(* Logix 5000 project; controller cal1615 1756-L62 rev 20.19; software revision 20.05; part 33 of 81 *)
(* tags used below, declared in another part *)
   FAULT : BOOL;   // Fault AFI
   p01_param_fan_zero_speed : REAL;
   p01_param_open_oven_recirc_sp : REAL;
   p01_recipe_active : recipe;   // Active Recipe
   p01_sys_scp : SYS_SCP;   // System Scaling
   p01r09_open_oven : BOOL;
   p01r09_pb_global_reset : BOOL;   // System Modes PB: Global Fault Reset
   p02_dint_from_hmi : hmi_dint;
   p11r02_shutdown_temp : BOOL;   // Zone 1 Misc Control Safe Shutdown Temperature
   p11r30 : routine;   // Zone 1 Temperature Control
   p12r02_shutdown_temp : BOOL;   // Zone 2 Misc Control Safe Shutdown Temperature
   p12r30 : routine;   // Zone 2 Temperature Control
   p13_ai_recirc_rpm : REAL;   // Zone 3 Analog Input Recirc Fan RPM
   p13_ao_recirc_selected_speed : REAL;   // Zone 3 Analog Output Recirc Fan VFD Selected Speed
   p13_di_recirc : acs800_di_normal;   // Zone 3 Digital Inputs Recirc Fan
   p13_di_recirc_fan_mtr_ts : BOOL;   // Zone 3 Digital Input Recirc Fan Motor Thermostat OK
   p13_di_recirc_flow_ok : BOOL;   // Zone 3 Digital Input Recirc Flow OK
   p13_dint_to_hmi : DINT[16];   // Zone 3 Temperature Control VFDs On
   p13_do_recirc : acs800_do_normal;   // Zone 3 Digital Outputs Supply Fan
   p13r01 : routine;   // Zone 3 Main
   p13r02_shutdown_temp : BOOL;   // Zone 3 Misc Control Safe Shutdown Temperature
   p13r20_state : DINT;   // Zone 3 Temperature Control State
   p13r32 : routine;   // Zone 3 Recirc VFD
   p13r32_pb_start : BOOL;   // Zone 3 Recirc VFD PB: Start
   p13r32_pb_stop : BOOL;   // Zone 3 Recirc VFD PB: Stop
   p13r32_request_auto_run : BOOL;   // Zone 3 Recirc Fan Run Request
   p13r32_run_permissive : BOOL;   // Zone 3 Recirc VFD Run Permissive
   p13r32_timer_fault : TIMER[5];   // Zone 3 Recirc VFD Fault Timer
   p13r32_timer_warning : TIMER[5];   // Zone 3 Supply VFD Warning Timer
   p13r32_vfd_stopped : BOOL;   // Zone 3 Recirc VFD VFD Stopped
   p19_ai_prs : REAL;   // Advanced Cooling Analog Input Pressure [PSI]
   p19_ai_tc01 : REAL;   // Advanced Cooling Analog Input Control Temperature 1
   p19_di_pump : BOOL;
   p19_di_tc01_bo : BOOL;   // Advanced Cooling Digital Input Control Thermocouple 1 Failure
   p19_di_tc02_bo : BOOL;   // Advanced Cooling Digital Input Control Thermocouple 2 Failure
   p19_dint_to_hmi : DINT[16];
   p19_param_tc01z : REAL;   // Advanced Cooling Parameter Control Temperature 1 Zero Offset
   p19r01 : routine;   // Advanced Cooling Main
   p19r02 : routine;   // Advanced Cooling Misc Control
   p19r02_fault_exists : BOOL;
   p19r02_timer_fault : TIMER[4];   // Advanced Cooling Misc Control Fault Delay
   p19r02_timer_warning : TIMER[4];   // Advanced Cooling Warning Delay
   p19r02_unack_fault : BOOL;   // Advanced Cooling Misc Control Unacknowledged Fault
   p19r02_unack_warning : BOOL;   // Advanced Cooling Misc Control Unacknowledged Warning
   p19r02_warning_exists : BOOL;
   p19r03 : routine;   // Advanced Cooling Input
   p19r03_prs_input_max : REAL;
   p19r03_prs_input_min : REAL;
   p19r03_prs_output_max : REAL;
   p19r03_prs_output_min : REAL;
   p19r03_timer_fault : TIMER[4];   // Advanced Cooling Input
   p19r03_timer_warning : TIMER[4];   // Advanced Cooling Input
   p19r04 : routine;   // Advanced Cooling Output
   p19r05 : routine;   // Advanced Cooling Dint to HMI
   p19r06 : routine;   // Advanced Cooling Real to HMI
   p19r07 : routine;   // Advanced Cooling Alarms
   p19r08 : routine;   // Advanced Cooling Warnings
   p19r09 : routine;   // Advanced Cooling Modes
   p19r10 : routine;   // Advanced Cooling Parameters
   p19r30 : routine;   // Advanced Cooling Temperature Control
   p19r31 : routine;   // Advanced Cooling Pump
   p23r02 : routine;   // Impreg Misc Control
(* P13_Zone_3, continued *)

ROUTINE R32_Recirc_VFD   (* ladder *)
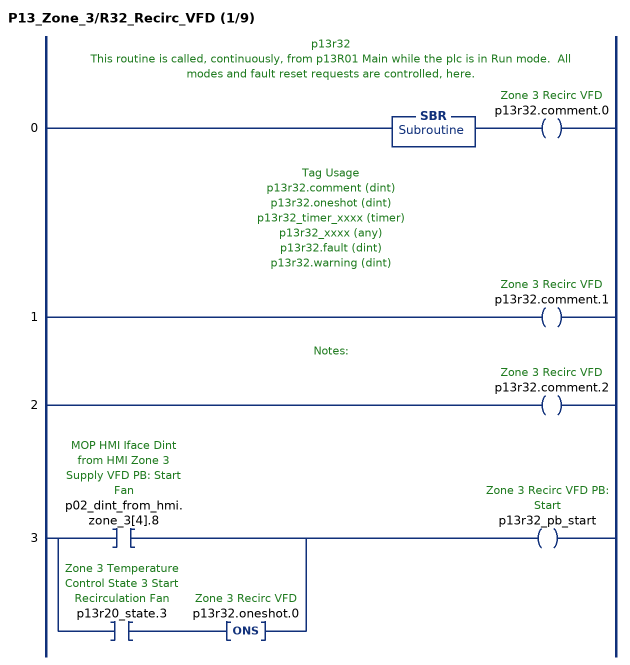
   // p13r32
   // This routine is called, continuously, from p13R01 Main while the plc is in Run mode.  All modes and fault reset requests are controlled, here.
   0: SBR()OTE(p13r32.comment.0);
   // Tag Usage
   // p13r32.comment (dint)
   // p13r32.oneshot (dint)
   // p13r32_timer_xxxx (timer)
   // p13r32_xxxx (any)
   // p13r32.fault (dint)
   // p13r32.warning (dint)
   1: OTE(p13r32.comment.1);
   // Notes:
   2: OTE(p13r32.comment.2);
   3: [XIC(p02_dint_from_hmi.zone_3[4].8) ,XIC(p13r20_state.3) ONS(p13r32.oneshot.0) ]OTE(p13r32_pb_start);
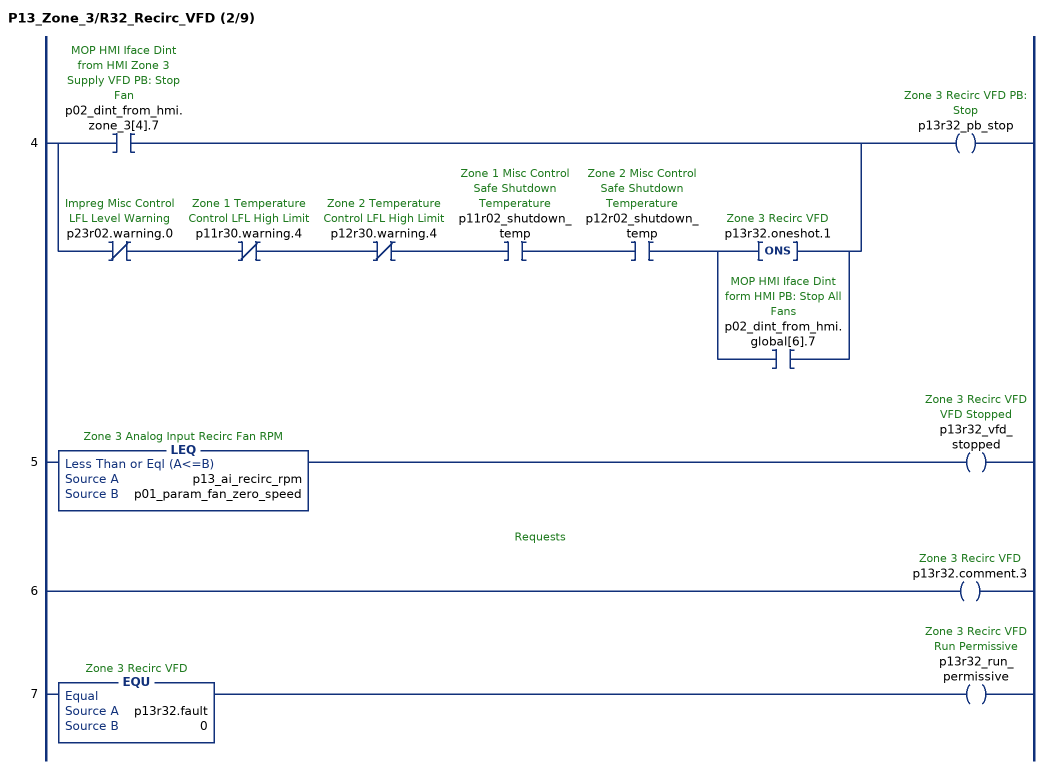
   4: [XIC(p02_dint_from_hmi.zone_3[4].7) ,XIO(p23r02.warning.0) XIO(p11r30.warning.4) XIO(p12r30.warning.4) XIC(p11r02_shutdown_temp) XIC(p12r02_shutdown_temp) [ONS(p13r32.oneshot.1) ,XIC(p02_dint_from_hmi.global[6].7) ] ]OTE(p13r32_pb_stop);
   5: LEQ(p13_ai_recirc_rpm,p01_param_fan_zero_speed)OTE(p13r32_vfd_stopped);
   // Requests
   6: OTE(p13r32.comment.3);
   7: EQU(p13r32.fault,0)OTE(p13r32_run_permissive);
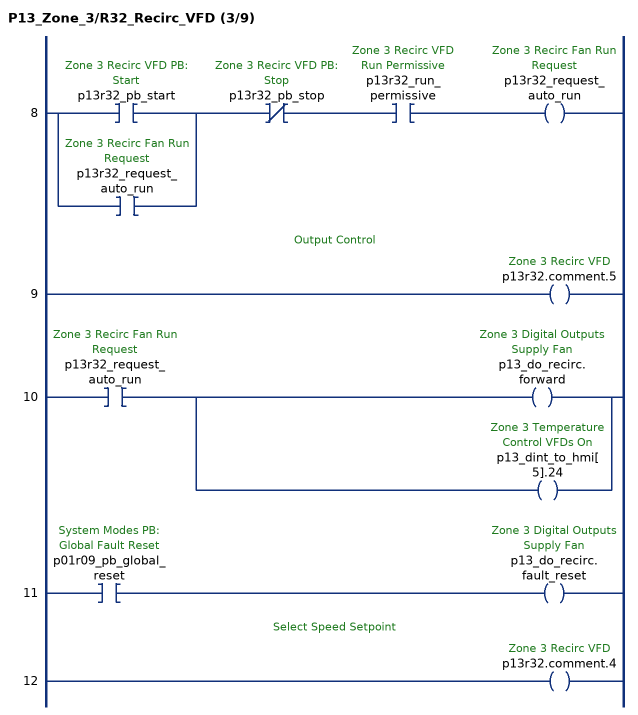
   8: [XIC(p13r32_pb_start) ,XIC(p13r32_request_auto_run) ]XIO(p13r32_pb_stop)XIC(p13r32_run_permissive)OTE(p13r32_request_auto_run);
   // Output Control
   9: OTE(p13r32.comment.5);
   10: XIC(p13r32_request_auto_run)[OTE(p13_do_recirc.forward) ,OTE(p13_dint_to_hmi[5].24) ];
   11: XIC(p01r09_pb_global_reset)OTE(p13_do_recirc.fault_reset);
   // Select Speed Setpoint
   12: OTE(p13r32.comment.4);
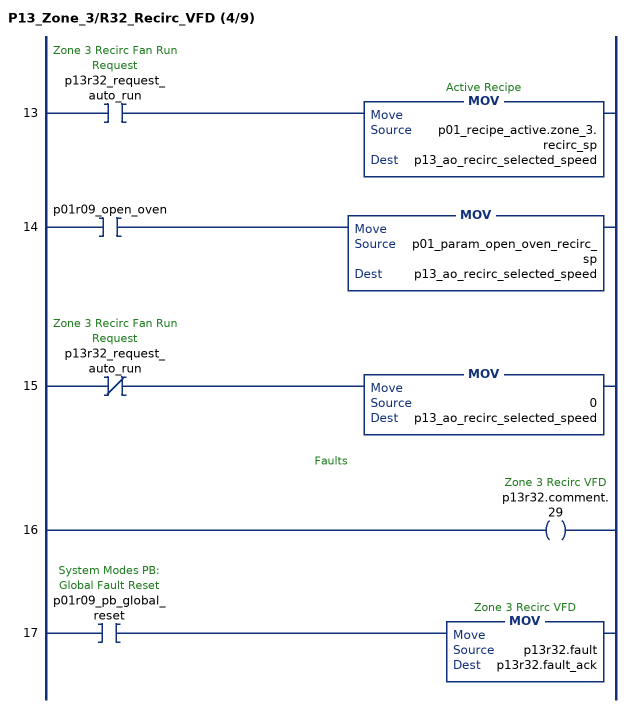
   13: XIC(p13r32_request_auto_run)MOV(p01_recipe_active.zone_3.recirc_sp,p13_ao_recirc_selected_speed);
   14: XIC(p01r09_open_oven)MOV(p01_param_open_oven_recirc_sp,p13_ao_recirc_selected_speed);
   15: XIO(p13r32_request_auto_run)MOV(0,p13_ao_recirc_selected_speed);
   // Faults
   16: OTE(p13r32.comment.29);
   17: XIC(p01r09_pb_global_reset)MOV(p13r32.fault,p13r32.fault_ack);
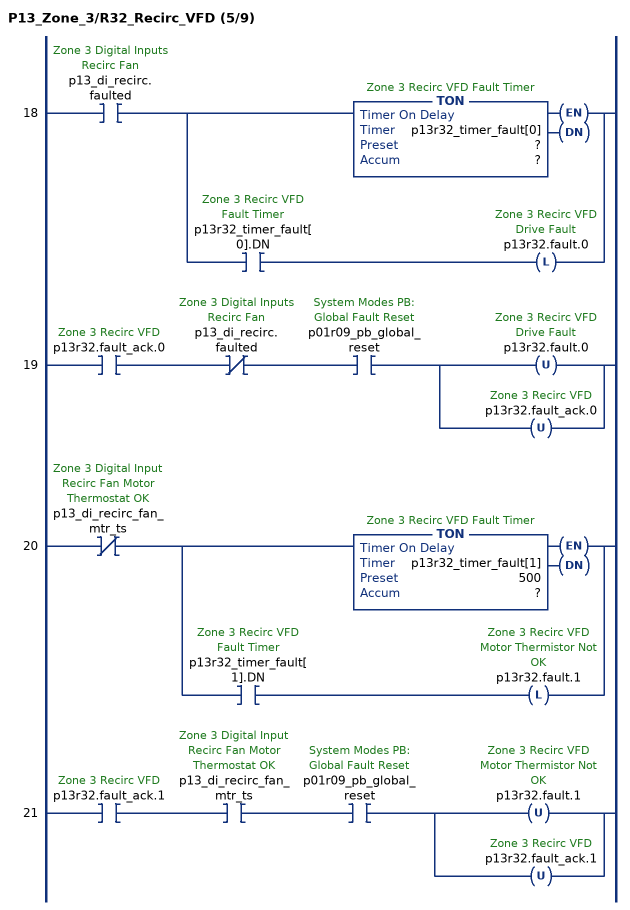
   18: XIC(p13_di_recirc.faulted)[TON(p13r32_timer_fault[0],?,?) ,XIC(p13r32_timer_fault[0].DN) OTL(p13r32.fault.0) ];
   19: XIC(p13r32.fault_ack.0)XIO(p13_di_recirc.faulted)XIC(p01r09_pb_global_reset)[OTU(p13r32.fault.0) ,OTU(p13r32.fault_ack.0) ];
   20: XIO(p13_di_recirc_fan_mtr_ts)[TON(p13r32_timer_fault[1],?,?) ,XIC(p13r32_timer_fault[1].DN) OTL(p13r32.fault.1) ];
   21: XIC(p13r32.fault_ack.1)XIC(p13_di_recirc_fan_mtr_ts)XIC(p01r09_pb_global_reset)[OTU(p13r32.fault.1) ,OTU(p13r32.fault_ack.1) ];
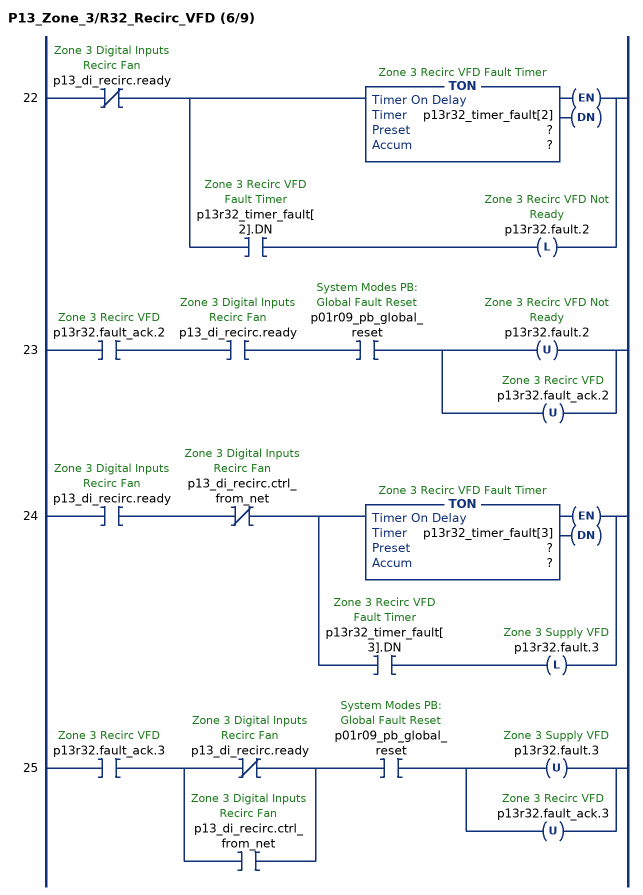
   22: XIO(p13_di_recirc.ready)[TON(p13r32_timer_fault[2],?,?) ,XIC(p13r32_timer_fault[2].DN) OTL(p13r32.fault.2) ];
   23: XIC(p13r32.fault_ack.2)XIC(p13_di_recirc.ready)XIC(p01r09_pb_global_reset)[OTU(p13r32.fault.2) ,OTU(p13r32.fault_ack.2) ];
   24: XIC(p13_di_recirc.ready)XIO(p13_di_recirc.ctrl_from_net)[TON(p13r32_timer_fault[3],?,?) ,XIC(p13r32_timer_fault[3].DN) OTL(p13r32.fault.3) ];
   25: XIC(p13r32.fault_ack.3)[XIO(p13_di_recirc.ready) ,XIC(p13_di_recirc.ctrl_from_net) ]XIC(p01r09_pb_global_reset)[OTU(p13r32.fault.3) ,OTU(p13r32.fault_ack.3) ];
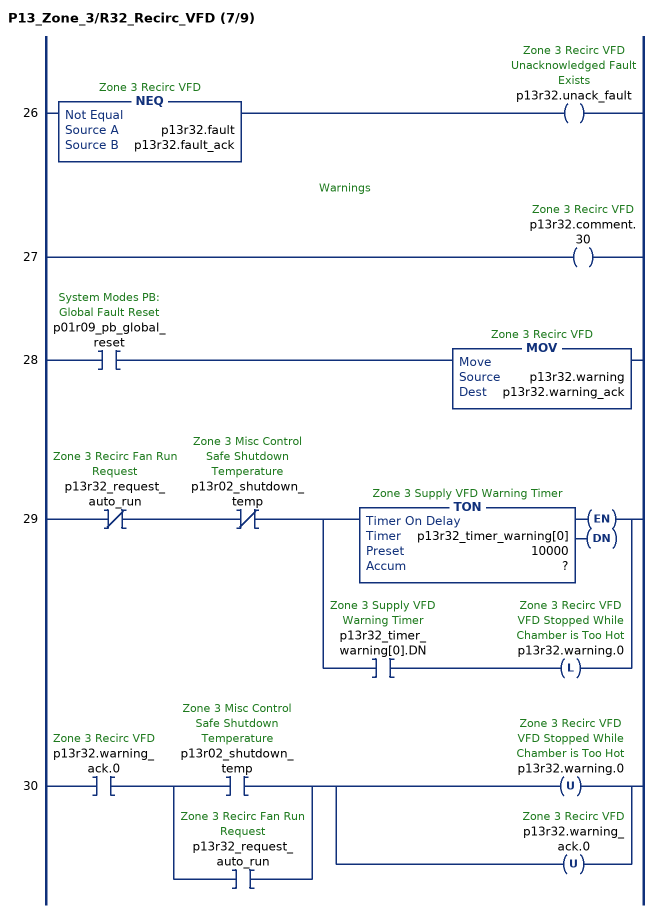
   26: NEQ(p13r32.fault,p13r32.fault_ack)OTE(p13r32.unack_fault);
   // Warnings
   27: OTE(p13r32.comment.30);
   28: XIC(p01r09_pb_global_reset)MOV(p13r32.warning,p13r32.warning_ack);
   29: XIO(p13r32_request_auto_run)XIO(p13r02_shutdown_temp)[TON(p13r32_timer_warning[0],?,?) ,XIC(p13r32_timer_warning[0].DN) OTL(p13r32.warning.0) ];
   30: XIC(p13r32.warning_ack.0)[XIC(p13r02_shutdown_temp) ,XIC(p13r32_request_auto_run) ][OTU(p13r32.warning.0) ,OTU(p13r32.warning_ack.0) ];
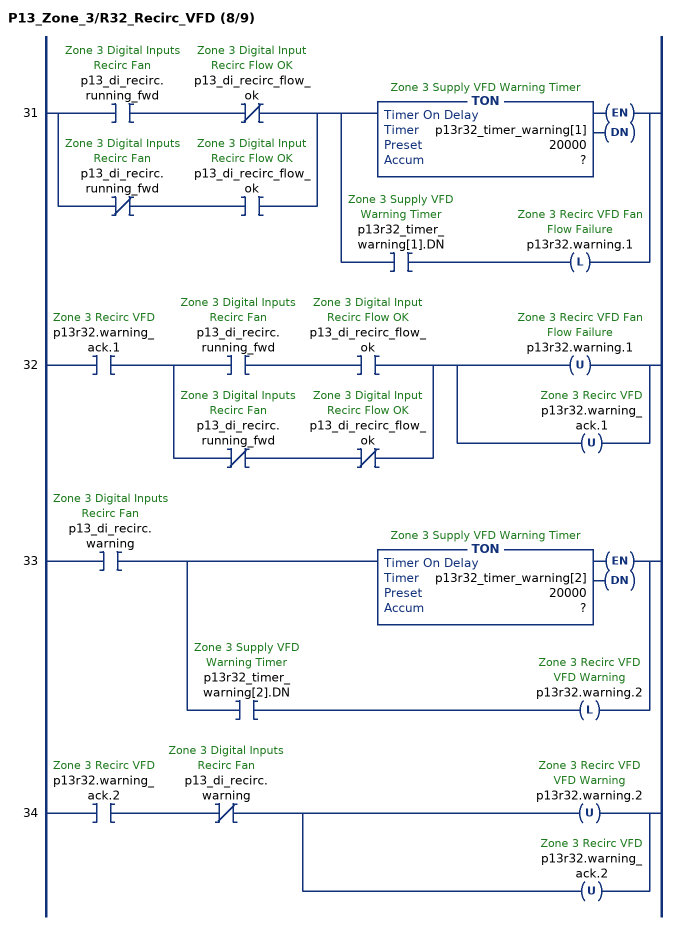
   31: [XIC(p13_di_recirc.running_fwd) XIO(p13_di_recirc_flow_ok) ,XIO(p13_di_recirc.running_fwd) XIC(p13_di_recirc_flow_ok) ][TON(p13r32_timer_warning[1],?,?) ,XIC(p13r32_timer_warning[1].DN) OTL(p13r32.warning.1) ];
   32: XIC(p13r32.warning_ack.1)[XIC(p13_di_recirc.running_fwd) XIC(p13_di_recirc_flow_ok) ,XIO(p13_di_recirc.running_fwd) XIO(p13_di_recirc_flow_ok) ][OTU(p13r32.warning.1) ,OTU(p13r32.warning_ack.1) ];
   33: XIC(p13_di_recirc.warning)[TON(p13r32_timer_warning[2],?,?) ,XIC(p13r32_timer_warning[2].DN) OTL(p13r32.warning.2) ];
   34: XIC(p13r32.warning_ack.2)XIO(p13_di_recirc.warning)[OTU(p13r32.warning.2) ,OTU(p13r32.warning_ack.2) ];
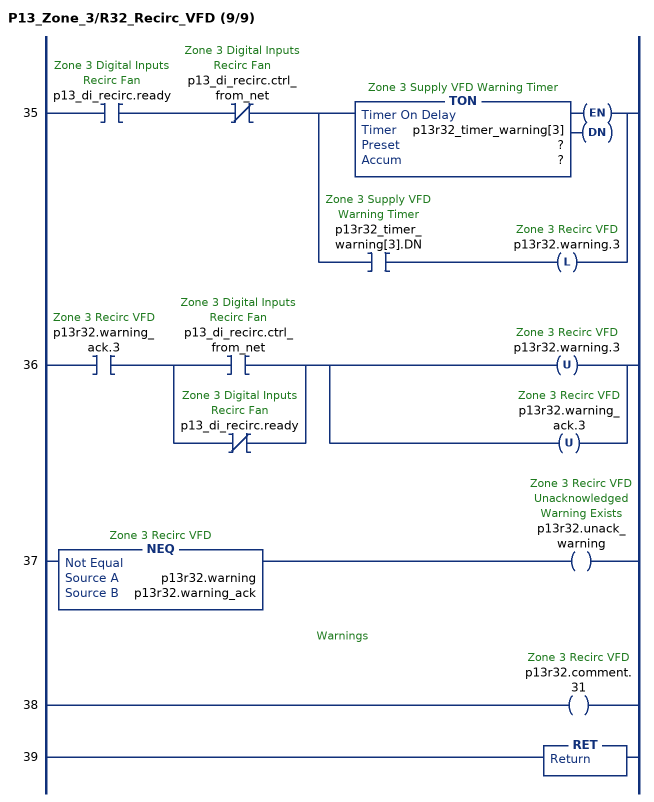
   35: XIC(p13_di_recirc.ready)XIO(p13_di_recirc.ctrl_from_net)[TON(p13r32_timer_warning[3],?,?) ,XIC(p13r32_timer_warning[3].DN) OTL(p13r32.warning.3) ];
   36: XIC(p13r32.warning_ack.3)[XIC(p13_di_recirc.ctrl_from_net) ,XIO(p13_di_recirc.ready) ][OTU(p13r32.warning.3) ,OTU(p13r32.warning_ack.3) ];
   37: NEQ(p13r32.warning,p13r32.warning_ack)OTE(p13r32.unack_warning);
   // Warnings
   38: OTE(p13r32.comment.31);
   39: RET();
END_ROUTINE
END_PROGRAM

PROGRAM P19_Advanced_Cooling   (* main routine R01_Main *)

ROUTINE R01_Main   (* ladder *)
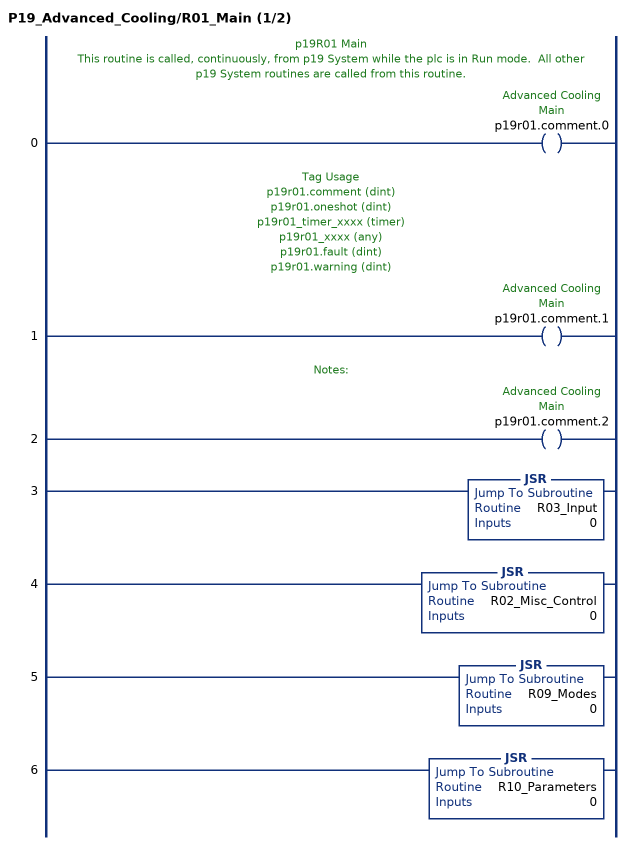
   // p19R01 Main
   // This routine is called, continuously, from p19 System while the plc is in Run mode.  All other p19 System routines are called from this routine.
   0: OTE(p19r01.comment.0);
   // Tag Usage
   // p19r01.comment (dint)
   // p19r01.oneshot (dint)
   // p19r01_timer_xxxx (timer)
   // p19r01_xxxx (any)
   // p19r01.fault (dint)
   // p19r01.warning (dint)
   1: OTE(p19r01.comment.1);
   // Notes:
   2: OTE(p19r01.comment.2);
   3: JSR(R03_Input,0);
   4: JSR(R02_Misc_Control,0);
   5: JSR(R09_Modes,0);
   6: JSR(R10_Parameters,0);
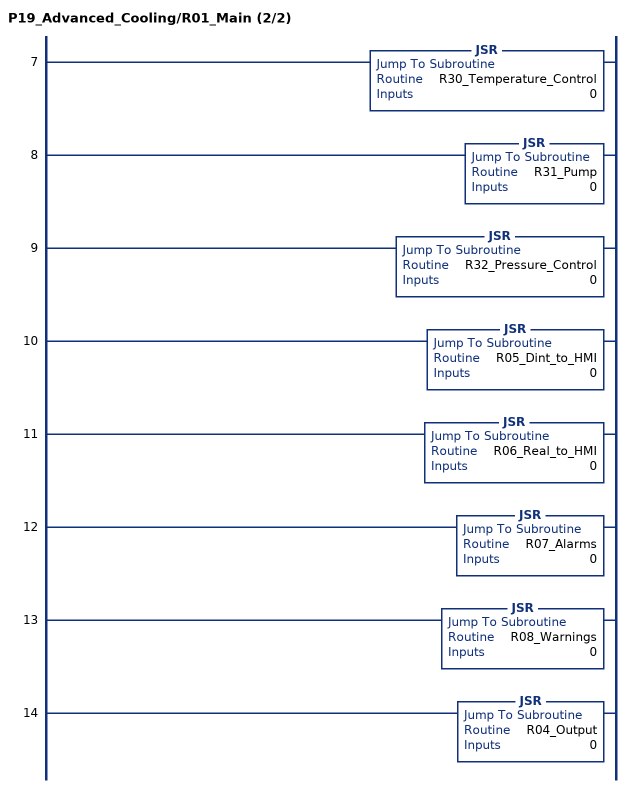
   7: JSR(R30_Temperature_Control,0);
   8: JSR(R31_Pump,0);
   9: JSR(R32_Pressure_Control,0);
   10: JSR(R05_Dint_to_HMI,0);
   11: JSR(R06_Real_to_HMI,0);
   12: JSR(R07_Alarms,0);
   13: JSR(R08_Warnings,0);
   14: JSR(R04_Output,0);
END_ROUTINE

ROUTINE R02_Misc_Control   (* ladder *)
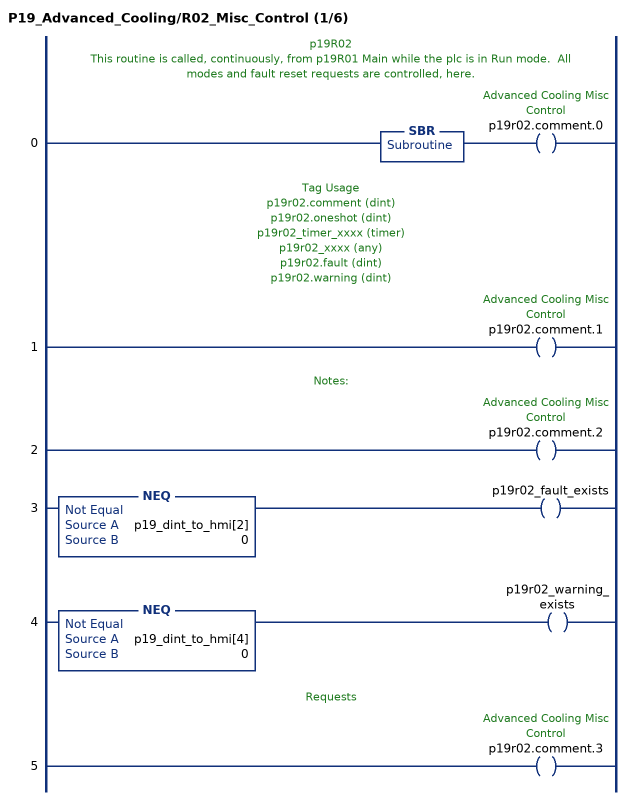
   // p19R02
   // This routine is called, continuously, from p19R01 Main while the plc is in Run mode.  All modes and fault reset requests are controlled, here.
   0: SBR()OTE(p19r02.comment.0);
   // Tag Usage
   // p19r02.comment (dint)
   // p19r02.oneshot (dint)
   // p19r02_timer_xxxx (timer)
   // p19r02_xxxx (any)
   // p19r02.fault (dint)
   // p19r02.warning (dint)
   1: OTE(p19r02.comment.1);
   // Notes:
   2: OTE(p19r02.comment.2);
   3: NEQ(p19_dint_to_hmi[2],0)OTE(p19r02_fault_exists);
   4: NEQ(p19_dint_to_hmi[4],0)OTE(p19r02_warning_exists);
   // Requests
   5: OTE(p19r02.comment.3);
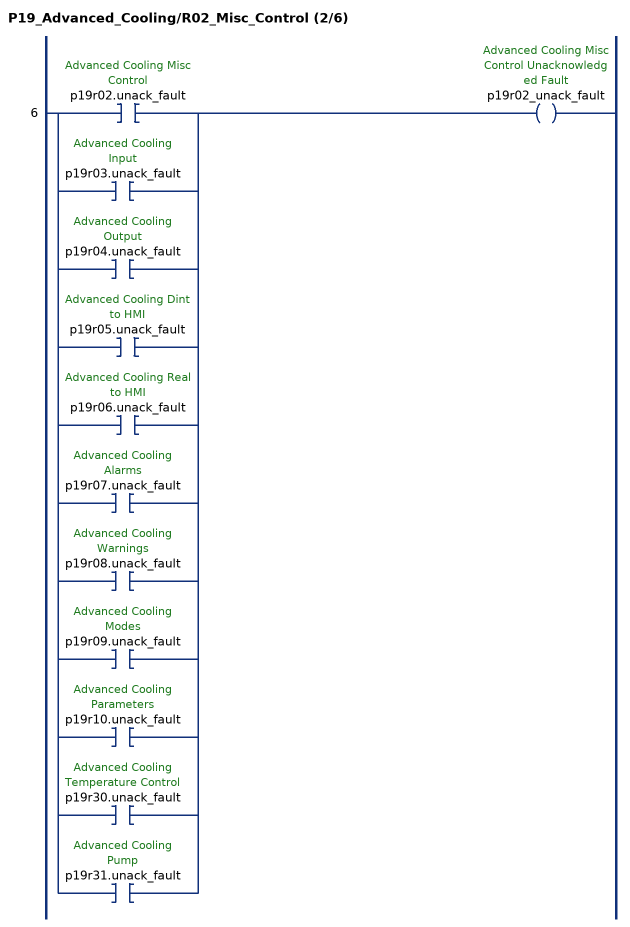
   6: [XIC(p19r02.unack_fault) ,XIC(p19r03.unack_fault) ,XIC(p19r04.unack_fault) ,XIC(p19r05.unack_fault) ,XIC(p19r06.unack_fault) ,XIC(p19r07.unack_fault) ,XIC(p19r08.unack_fault) ,XIC(p19r09.unack_fault) ,XIC(p19r10.unack_fault) ,XIC(p19r30.unack_fault) ,XIC(p19r31.unack_fault) ]OTE(p19r02_unack_fault);
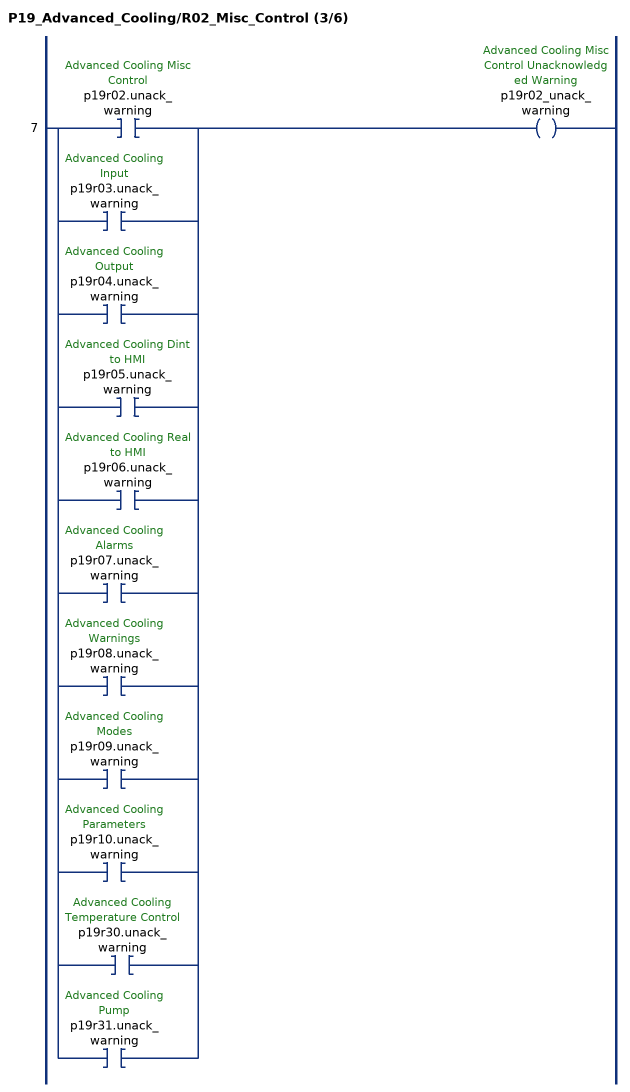
   7: [XIC(p19r02.unack_warning) ,XIC(p19r03.unack_warning) ,XIC(p19r04.unack_warning) ,XIC(p19r05.unack_warning) ,XIC(p19r06.unack_warning) ,XIC(p19r07.unack_warning) ,XIC(p19r08.unack_warning) ,XIC(p19r09.unack_warning) ,XIC(p19r10.unack_warning) ,XIC(p19r30.unack_warning) ,XIC(p19r31.unack_warning) ]OTE(p19r02_unack_warning);
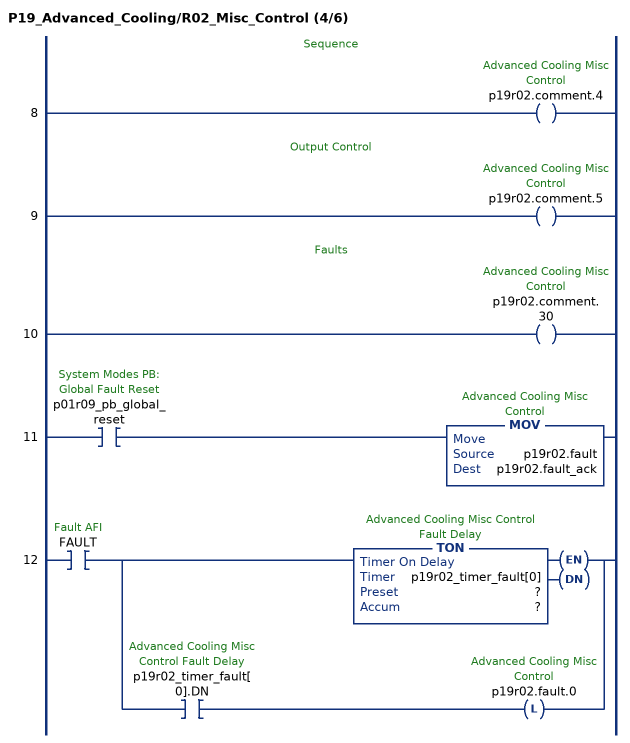
   // Sequence
   8: OTE(p19r02.comment.4);
   // Output Control
   9: OTE(p19r02.comment.5);
   // Faults
   10: OTE(p19r02.comment.30);
   11: XIC(p01r09_pb_global_reset)MOV(p19r02.fault,p19r02.fault_ack);
   12: XIC(FAULT)[TON(p19r02_timer_fault[0],?,?) ,XIC(p19r02_timer_fault[0].DN) OTL(p19r02.fault.0) ];
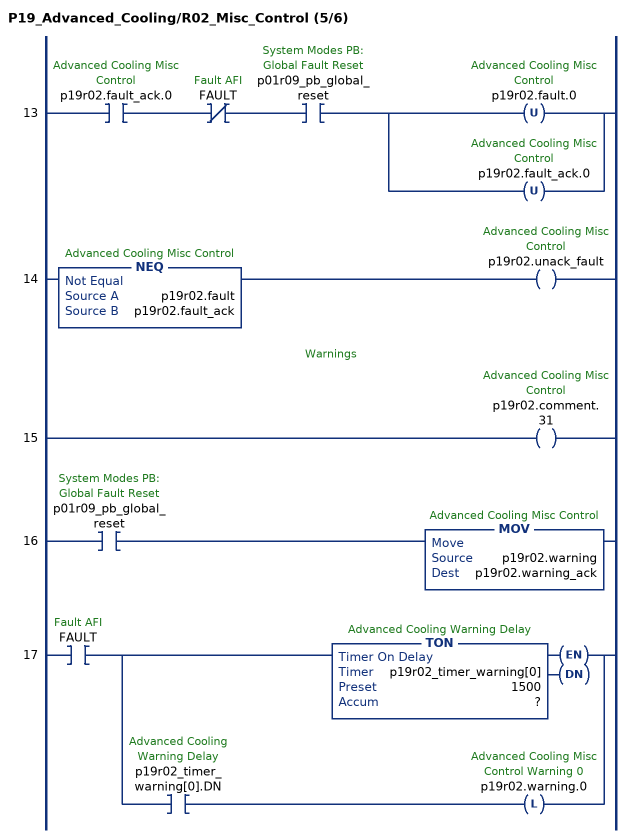
   13: XIC(p19r02.fault_ack.0)XIO(FAULT)XIC(p01r09_pb_global_reset)[OTU(p19r02.fault.0) ,OTU(p19r02.fault_ack.0) ];
   14: NEQ(p19r02.fault,p19r02.fault_ack)OTE(p19r02.unack_fault);
   // Warnings
   15: OTE(p19r02.comment.31);
   16: XIC(p01r09_pb_global_reset)MOV(p19r02.warning,p19r02.warning_ack);
   17: XIC(FAULT)[TON(p19r02_timer_warning[0],?,?) ,XIC(p19r02_timer_warning[0].DN) OTL(p19r02.warning.0) ];
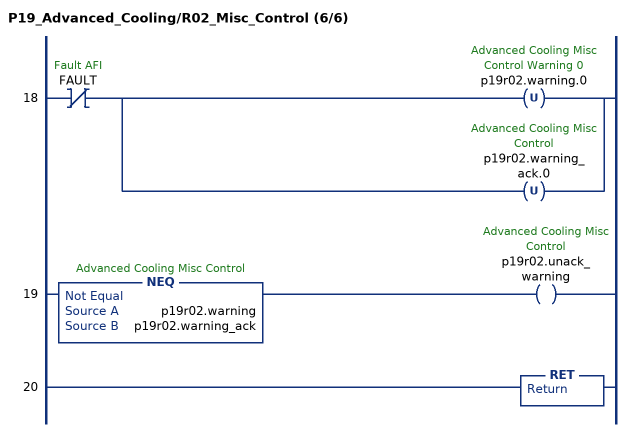
   18: XIO(FAULT)[OTU(p19r02.warning.0) ,OTU(p19r02.warning_ack.0) ];
   19: NEQ(p19r02.warning,p19r02.warning_ack)OTE(p19r02.unack_warning);
   20: RET();
END_ROUTINE

ROUTINE R03_Input   (* ladder *)
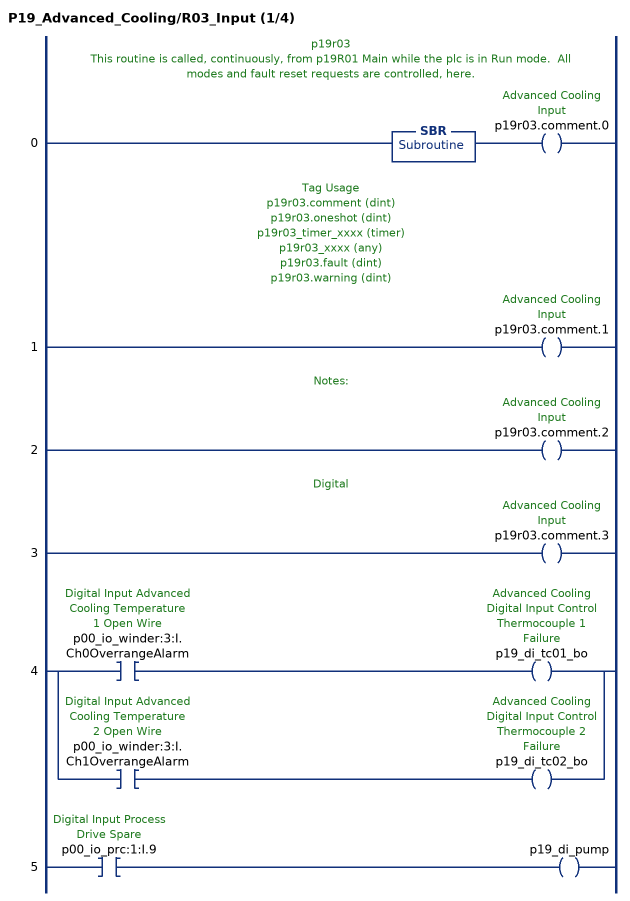
   // p19r03
   // This routine is called, continuously, from p19R01 Main while the plc is in Run mode.  All modes and fault reset requests are controlled, here.
   0: SBR()OTE(p19r03.comment.0);
   // Tag Usage
   // p19r03.comment (dint)
   // p19r03.oneshot (dint)
   // p19r03_timer_xxxx (timer)
   // p19r03_xxxx (any)
   // p19r03.fault (dint)
   // p19r03.warning (dint)
   1: OTE(p19r03.comment.1);
   // Notes:
   2: OTE(p19r03.comment.2);
   // Digital
   3: OTE(p19r03.comment.3);
   4: [XIC(p00_io_winder:3:I.Ch0OverrangeAlarm) OTE(p19_di_tc01_bo) ,XIC(p00_io_winder:3:I.Ch1OverrangeAlarm) OTE(p19_di_tc02_bo) ];
   5: XIC(p00_io_prc:1:I.9)OTE(p19_di_pump);
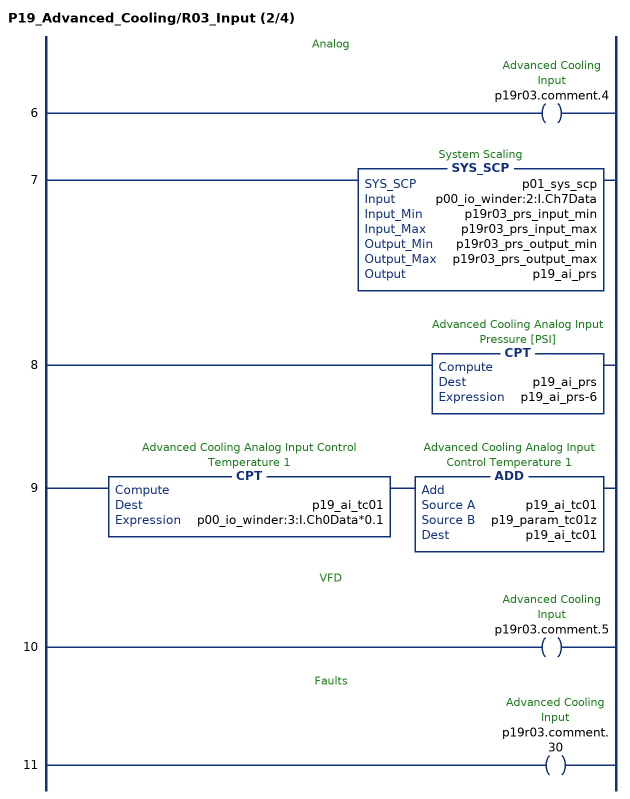
   // Analog
   6: OTE(p19r03.comment.4);
   7: SYS_SCP(p01_sys_scp,p00_io_winder:2:I.Ch7Data,p19r03_prs_input_min,p19r03_prs_input_max,p19r03_prs_output_min,p19r03_prs_output_max,p19_ai_prs);
   8: CPT(p19_ai_prs,p19_ai_prs-6);
   9: CPT(p19_ai_tc01,p00_io_winder:3:I.Ch0Data*0.1)ADD(p19_ai_tc01,p19_param_tc01z,p19_ai_tc01);
   // VFD
   10: OTE(p19r03.comment.5);
   // Faults
   11: OTE(p19r03.comment.30);
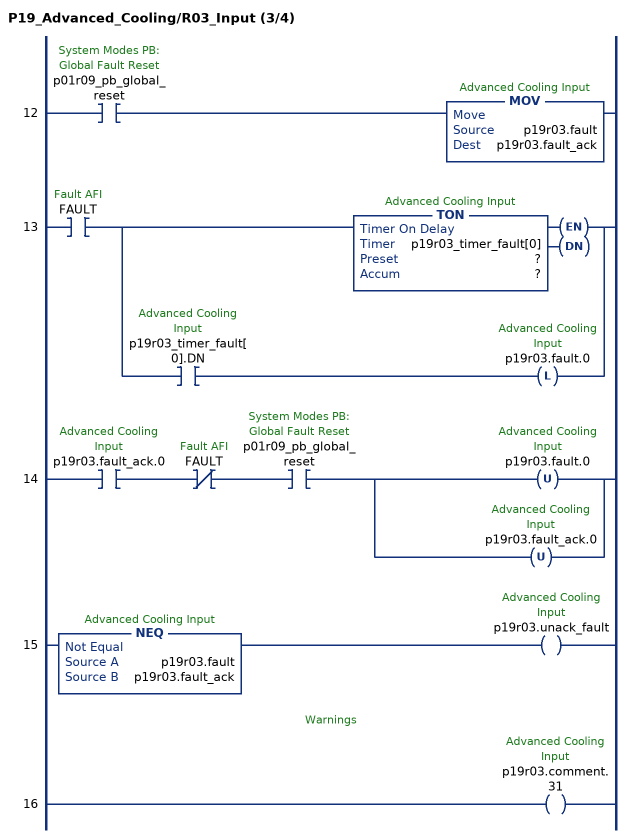
   12: XIC(p01r09_pb_global_reset)MOV(p19r03.fault,p19r03.fault_ack);
   13: XIC(FAULT)[TON(p19r03_timer_fault[0],?,?) ,XIC(p19r03_timer_fault[0].DN) OTL(p19r03.fault.0) ];
   14: XIC(p19r03.fault_ack.0)XIO(FAULT)XIC(p01r09_pb_global_reset)[OTU(p19r03.fault.0) ,OTU(p19r03.fault_ack.0) ];
   15: NEQ(p19r03.fault,p19r03.fault_ack)OTE(p19r03.unack_fault);
   // Warnings
   16: OTE(p19r03.comment.31);
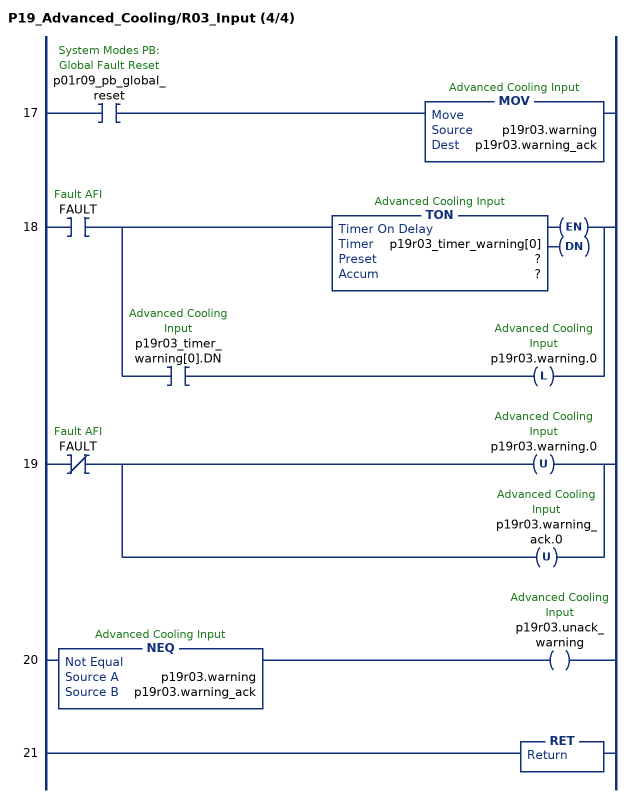
   17: XIC(p01r09_pb_global_reset)MOV(p19r03.warning,p19r03.warning_ack);
   18: XIC(FAULT)[TON(p19r03_timer_warning[0],?,?) ,XIC(p19r03_timer_warning[0].DN) OTL(p19r03.warning.0) ];
   19: XIO(FAULT)[OTU(p19r03.warning.0) ,OTU(p19r03.warning_ack.0) ];
   20: NEQ(p19r03.warning,p19r03.warning_ack)OTE(p19r03.unack_warning);
   21: RET();
END_ROUTINE
